FUNCTION_BLOCK Plant
  (* Standard: 61499-2 *)
  (* Version 0.1, 2015-00-15, Th?o, PC_THEO *)
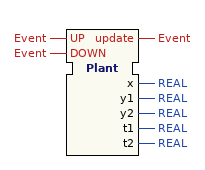
  EVENT_INPUT
    UP;
    DOWN;
  END_EVENT
  EVENT_OUTPUT
    update;
  END_EVENT
  VAR_OUTPUT
    x : REAL;
    y1 : REAL;
    y2 : REAL;
    t1 : REAL;
    t2 : REAL;
  END_VAR
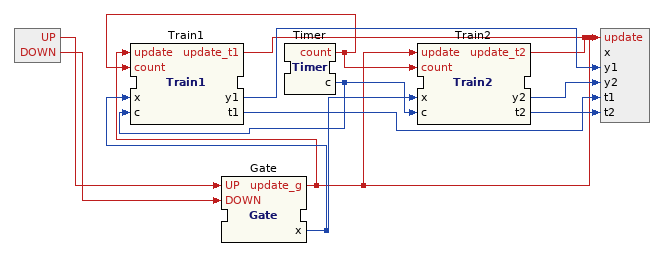
  FBS
    Train1 : Train1;
    Gate : Gate;
    Train2 : Train2;
    Timer : Timer;
  END_FBS
  EVENT_CONNECTIONS
    UP TO Gate.UP;
    DOWN TO Gate.DOWN;
    Train1.update_t1 TO update;
    Gate.update_g TO update;
    Train2.update_t2 TO update;
    Gate.update_g TO Train1.update;
    Gate.update_g TO Train2.update;
    Timer.count TO Train1.count;
    Timer.count TO Train2.count;
  END_CONNECTIONS
  DATA_CONNECTIONS
    Train1.y1 TO y1;
    Train2.y2 TO y2;
    Train1.t1 TO t1;
    Train2.t2 TO t2;
    Gate.x TO Train1.x;
    Gate.x TO Train2.x;
    Timer.c TO Train1.c;
    Timer.c TO Train2.c;
  END_CONNECTIONS
END_FUNCTION_BLOCK
